SUBAPPLICATION Klappen (* Subapplication Type *)
  (* Standard: 61499-2 *)
  (* Version 1.0, 2023-01-29, Franz *)
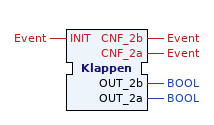
  EVENT_INPUT
    INIT;
  END_EVENT
  EVENT_OUTPUT
    CNF_2b;
    CNF_2a;
  END_EVENT
  VAR_OUTPUT
    OUT_2b : BOOL;
    OUT_2a : BOOL;
  END_VAR
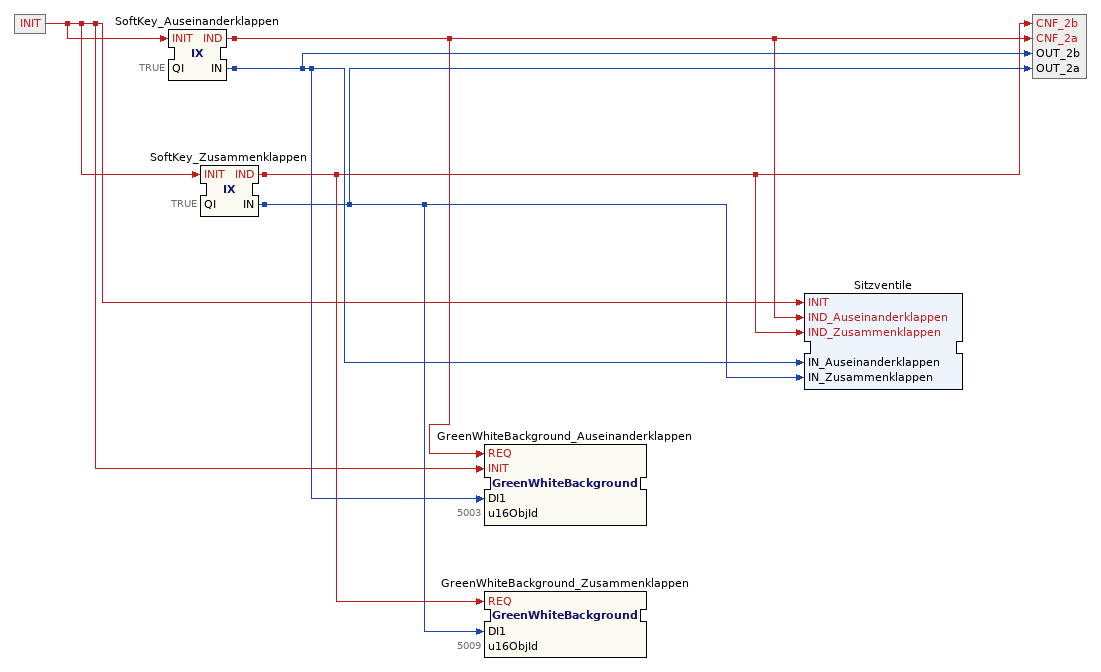
  FBS
    SoftKey_Auseinanderklappen : IX(QI := TRUE);
    GreenWhiteBackground_Auseinanderklappen : GreenWhiteBackground(u16ObjId := 5003);
    SoftKey_Zusammenklappen : IX(QI := TRUE);
    GreenWhiteBackground_Zusammenklappen : GreenWhiteBackground(u16ObjId := 5009);
  END_FBS
  SUBAPPLICATION Sitzventile (* Sitzventile *)
    EVENT_INPUT
      INIT;
      IND_Auseinanderklappen;
      IND_Zusammenklappen;
    END_EVENT
    VAR_INPUT
      IN_Auseinanderklappen : BOOL;
      IN_Zusammenklappen : BOOL;
    END_VAR
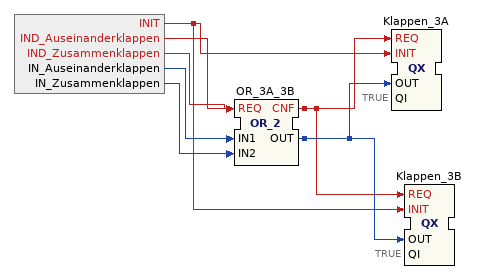
    FBS
      Klappen_3B : QX(QI := TRUE);
      Klappen_3A : QX(QI := TRUE);
      OR_3A_3B : OR_2; {SET_ATTRIBUTE(PinComment, IN1:Auseinanderklappen)} {SET_ATTRIBUTE(PinComment, IN2:Zusammenklappen)}
    END_FBS
    EVENT_CONNECTIONS
      OR_3A_3B.CNF TO Klappen_3B.REQ;
      OR_3A_3B.CNF TO Klappen_3A.REQ;
      INIT TO Klappen_3B.INIT;
      INIT TO Klappen_3A.INIT;
      IND_Auseinanderklappen TO OR_3A_3B.REQ;
      IND_Zusammenklappen TO OR_3A_3B.REQ;
    END_CONNECTIONS
    DATA_CONNECTIONS
      OR_3A_3B.OUT TO Klappen_3B.OUT;
      OR_3A_3B.OUT TO Klappen_3A.OUT;
      IN_Auseinanderklappen TO OR_3A_3B.IN1;
      IN_Zusammenklappen TO OR_3A_3B.IN2;
    END_CONNECTIONS
  END_SUBAPPLICATION
  EVENT_CONNECTIONS
    SoftKey_Auseinanderklappen.IND TO GreenWhiteBackground_Auseinanderklappen.REQ;
    INIT TO SoftKey_Auseinanderklappen.INIT;
    SoftKey_Auseinanderklappen.IND TO CNF_2b;
    INIT TO SoftKey_Zusammenklappen.INIT;
    SoftKey_Zusammenklappen.IND TO CNF_2a;
    INIT TO GreenWhiteBackground_Auseinanderklappen.INIT;
    INIT TO Sitzventile.INIT;
    SoftKey_Auseinanderklappen.IND TO Sitzventile.IND_Auseinanderklappen;
    SoftKey_Zusammenklappen.IND TO Sitzventile.IND_Zusammenklappen;
    SoftKey_Zusammenklappen.IND TO GreenWhiteBackground_Zusammenklappen.REQ;
  END_CONNECTIONS
  DATA_CONNECTIONS
    SoftKey_Auseinanderklappen.IN TO GreenWhiteBackground_Auseinanderklappen.DI1;
    SoftKey_Auseinanderklappen.IN TO OUT_2b;
    SoftKey_Zusammenklappen.IN TO OUT_2a;
    SoftKey_Auseinanderklappen.IN TO Sitzventile.IN_Auseinanderklappen;
    SoftKey_Zusammenklappen.IN TO Sitzventile.IN_Zusammenklappen;
    SoftKey_Zusammenklappen.IN TO GreenWhiteBackground_Zusammenklappen.DI1;
  END_CONNECTIONS
END_SUBAPPLICATION
